{attribute addProperty BoxType "EK1100-0000-0018"}
{attribute addProperty Id "Beckhoff_EKx9xxEK1122Beckhoff_EKx9xxEK1122_226D7D504688586"}
{attribute addProperty CRC "3393617451"}
{attribute addProperty SizeInBites "4688"}
{attribute addProperty SizeInBytes "586"}
TYPE Beckhoff_EKx9xx_CA467E2B EXTENDS EK1100_179A0949 :
STRUCT
	{attribute addProperty Name "Beckhoff_EKx9xxEK1122"}
	Beckhoff_EKx9xxEK1122 : Beckhoff_EKx9xxEK1122_226D7D50;
END_STRUCT
END_TYPE

(* stored: Version 1.2.0.0, ProductVersion 3.1.4024.9
   DUT Beckhoff_EKx9xx_CA467E2B: Id {5d56a7cc-b438-4026-bcd9-5ec85663fe71} *)
